// TIA Portal V20 export
DATA_BLOCK "BK29"   // DB280
// stored: MemoryReserve 100
   VAR
      "SUCTION PAD TOP RIGHT VACUUM ON" : Bool := FALSE;
      "SUCTION PAD TOP RIGHT VACUUM OFF" : Bool := FALSE;
      "SUCTION PAD TOP LEFT VACUUM ON" : Bool := FALSE;
      "SUCTION PAD TOP LEFT VACUUM OFF" : Bool := FALSE;
      "SUCTION PAD BTM RIGHT VACUUM ON" : Bool := FALSE;
      "SUCTION PAD BTM RIGHT VACUUM OFF" : Bool := FALSE;
      "SUCTION PAD BTM LEFT VACUUM ON" : Bool := FALSE;
      "SUCTION PAD BTM LEFT VACUUM OFF" : Bool := FALSE;
   END_VAR
BEGIN
END_DATA_BLOCK
